% RSLogix 500 project PLC_1_L5-4.RSS, saved by version 12.00.00.00 %
PROJECT "UNTITLED"    % processor: Bul.1763 MicroLogix 1100 Series B %

PROGRAM FILES
  LAD 2   8 rungs

DATA FILES
  O0 OUTPUT  5 elements
  I1 INPUT  6 elements
  S2 STATUS  66 elements
  B3 BINARY  1 elements
  T4 TIMER  4 elements
  C5 COUNTER  1 elements
  R6 CONTROL  1 elements
  N7 INTEGER  1 elements
  F8 FLOAT  1 elements

LADDER 2
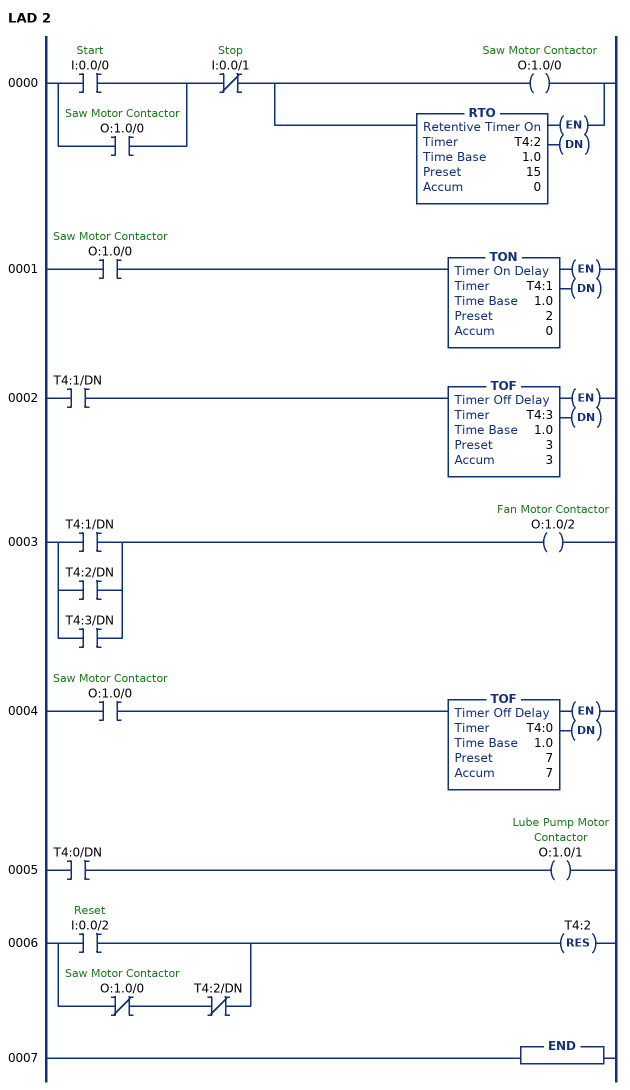
% Rung: 0 %
SOR BST XIC I:0.0/0 NXB XIC O:1.0/0 BND XIO I:0.0/1 BST OTE O:1.0/0 NXB RTO T4:2 1.0 15 0 BND EOR
%   I:0.0/0  "Start" %
%   O:1.0/0  "Saw Motor Contactor" %
%   I:0.0/1  "Stop" %
% Rung: 1 %
SOR XIC O:1.0/0 TON T4:1 1.0 2 0 EOR
%   O:1.0/0  "Saw Motor Contactor" %
% Rung: 2 %
SOR XIC T4:1/DN TOF T4:3 1.0 3 3 EOR
% Rung: 3 %
SOR BST XIC T4:1/DN NXB XIC T4:2/DN NXB XIC T4:3/DN BND OTE O:1.0/2 EOR
%   O:1.0/2  "Fan Motor Contactor" %
% Rung: 4 %
SOR XIC O:1.0/0 TOF T4:0 1.0 7 7 EOR
%   O:1.0/0  "Saw Motor Contactor" %
% Rung: 5 %
SOR XIC T4:0/DN OTE O:1.0/1 EOR
%   O:1.0/1  "Lube Pump Motor Contactor" %
% Rung: 6 %
SOR BST XIC I:0.0/2 NXB XIO O:1.0/0 XIO T4:2/DN BND RES T4:2 EOR
%   I:0.0/2  "Reset" %
%   O:1.0/0  "Saw Motor Contactor" %
% Rung: 7 %
SOR END EOR

DATA TABLE (non-zero values as saved)
DATA T4
% .PRE .ACC %
% T4:0 % 7 7
% T4:1 % 2 0
% T4:2 % 15 0
% T4:3 % 3 3
